{attribute 'qualified_only'}
VAR_GLOBAL
	// Schnittstellenvariablen 
		// System: 
		SystemState								:eSystemState; 
		SystemCommand							:eSystemCommand; 
		ErrorID									:INT;
		
		// Kontrollvariablen: 
		Reset									:BOOL;
		Execute									:BOOL;
		
		// Prozessvariablen
		eKraftLimitValue						:sKraftVariablen;
		eKraftErreichtValue						:sKraftVariablen;
		
		
		// SkillStates
		
		// ObjectStates
		Robot_State								:eObjectAktorState;
		Greifer_State							:eObjectAktorState;
		Sensor_State							:eObjectAktorState;
END_VAR

(* stored: Version 1.1.0.1
   GVL GVL: Id {935c66c4-3c1a-441a-babc-36b55c5306d6} *)
